FUNCTION_BLOCK FB_PID
(*Simple PID Controller*)

VAR_INPUT
	fSetpoint: LREAL; (*setpoint value*)
	fProcessVariable: LREAL; (*actual value*)
	fKp: LREAL; (*proportional gain-Kp*)
	fKi: LREAL; (*integral gain-Ki*)
	fKd: LREAL; (*derivative gain-Kd*)
	fCycleTime: LREAL; (*controller cycle time in seconds(s)*)
	fMaxOutput: LREAL; (*maximum output command*)
	fMinOutput: LREAL; (*minimum output command*)
	bReset: BOOL; (*reset flag*)
END_VAR

VAR_OUTPUT
	fOutput: LREAL; (*controller output command*)
END_VAR

VAR
	Error: LREAL := 0; (*error between setpoint and process variable*)
	Integral: LREAL := 0; (*accumulated error*)
	Derivative: LREAL := 0; (*error rate of change*)
	LastError: LREAL := 0; (*error on last execution*)
	CycleCount: INT := 0; (*execution cycle count*)
END_VAR

(*Reset PID calculations when requested*)
IF bReset THEN
	Error := 0;
	Integral := 0;
	Derivative := 0;
	LastError := 0;
END_IF

(*Calculate the error between the setpoint and the process variable*)
Error := fSetpoint - fProcessVariable;

(*Only allow integral component to contibute to the controller output when the error is fairly small. 
  This is done to prevent severe overshoot on startup due to the nature of temperature control with
  a single output (heat, but no cooling).*)
IF ABS(Error) < 10 THEN
	(*Calculate accumulated error scaled to controller cycle time*)
	Integral := Integral + (Error * fCycleTime);
ELSE
	Integral := 0;
END_IF

(*Calculate the error rate of change*)
Derivative := (Error - LastError)/fCycleTime;

(*Calculate the controller output command*)
fOutput := (fKp * Error) + (fKi * Integral) + (fKd * Derivative);

IF fOutput > fMaxOutput THEN
	fOutput := fMaxOutput;
END_IF
IF fOutput < fMinOutput THEN
	fOutput := fMinOutput;
END_IF

(*Store the current error for the next cycle*)
LastError := Error;

(*Reset controller components every 30 cycles in order to prevent integral component from running away.
  This is done to prevent severe overshoot due to the nature of temperature control with
  a single output (heat, but no cooling).*)
CycleCount := CycleCount + 1;
IF CycleCount >= 30 THEN
	Error := 0;
	Integral := 0;
	Derivative := 0;
	LastError := 0;
	CycleCount := 0;
END_IF

END_FUNCTION_BLOCK

(* stored: Version 1.1.0.1, ProductVersion 3.1.4020.12
   POU FB_PID: Id {9948b47d-b616-4fdc-9dcf-d79a24cdad0b}, SpecialFunc None *)
